Fanuc KAREL source: kt00928.KL

PROGRAM KT00928
%STACKSIZE=65535
%PRIORITY=65535
%NOLOCKGROUP
VAR
S1 : STRING[80]
S2 : STRING[80]
OUT : INTEGER
BEGIN
S1='A'
S2='B'
S1='A'
S2='B'
-- UNRESOLVED_PC line 12 opcodes [27 22 2A 27 9D 76 23] marker_code=56
END KT00928
